(* PLC project MotionTest1, Higen MCL 1 *)
(* stored: creationDateTime 2012-01-06T15:20:13, modificationDateTime 2013-07-14T17:27:56 *)

FUNCTION_BLOCK wxgetval
  VAR
    getpy : python_gear;
    latch : SR;
  END_VAR
  VAR_INPUT
    name : STRING;
  END_VAR
  VAR_OUTPUT
    val : BOOL;
  END_VAR
  VAR  (* added by the conversion: wires and edge detectors of the diagram *)
    _EQ41_ENO : BOOL;
    _EQ41_OUT : BOOL;
    _EQ3_ENO : BOOL;
    _EQ3_OUT : BOOL;
  END_VAR

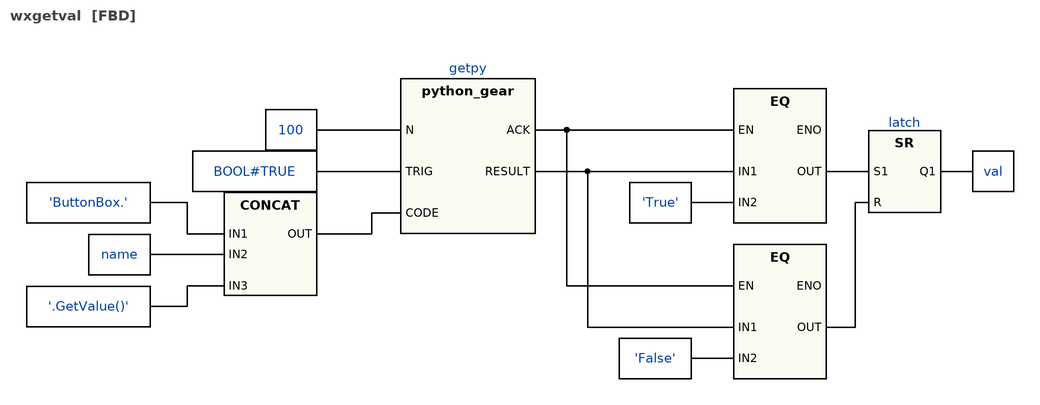
(* FBD diagram, written out as Structured Text *)
getpy(N := 100, TRIG := BOOL#TRUE, CODE := CONCAT('ButtonBox.', name, '.GetValue()'));
_EQ41_OUT := EQ(EN := getpy.ACK, IN1 := getpy.RESULT, IN2 := 'True', ENO => _EQ41_ENO);
_EQ3_OUT := EQ(EN := getpy.ACK, IN1 := getpy.RESULT, IN2 := 'False', ENO => _EQ3_ENO);
latch(S1 := _EQ41_OUT, R := _EQ3_OUT);
val := latch.Q1;
END_FUNCTION_BLOCK

(* -- *)
PROGRAM main
  VAR
    Done : BOOL;
    Axis : AXIS_REF;
    mPn : LREAL;
    mVn : LREAL;
    bt1 : wxgetval;
    Block1 : wxgetval;
    Block6 : wxgetval;
    MC_Sim0 : MC_Sim;
    MC_Power0 : MC_Power;
    MC_ReadActualPosition0 : MC_ReadActualPosition;
    MC_SetPosition0 : MC_SetPosition;
    MC_MoveAbsolute0 : MC_MoveAbsolute;
    Output : MC_OUTPUT_REF;
    OutputBits : DWORD;
    Track1 : BOOL;
    Track2 : BOOL;
    Track3 : BOOL;
    Velocity : LREAL := 1000.0;
    TrackList : MC_TRACK_REF;
    CamSwitchList : MC_CAMSWITCH_REF;
    MC_TRACK_REF_FROM_CSV0 : MC_TRACK_REF_FROM_CSV;
    MC_CAMSWITCH_REF_FROM_CSV0 : MC_CAMSWITCH_REF_FROM_CSV;
    MC_DigitalCamSwitch0 : MC_DigitalCamSwitch;
    MC_CreateOutput0 : MC_CreateOutput;
    MC_ReadActualVelocity0 : MC_ReadActualVelocity;
    MC_ReadOutputBits0 : MC_ReadOutputBits;
    MC_MoveAbsolute1 : MC_MoveAbsolute;
    MC_MoveAbsolute2 : MC_MoveAbsolute;
    MC_MoveAbsolute3 : MC_MoveAbsolute;
    MC_MoveAbsolute4 : MC_MoveAbsolute;
    MC_MoveAbsolute5 : MC_MoveAbsolute;
    MC_ReadOutputBit0 : MC_ReadOutputBit;
    MC_ReadOutputBit1 : MC_ReadOutputBit;
    MC_WriteParameter0 : MC_WriteParameter;
    MC_MoveAbsolute6 : MC_MoveAbsolute;
    MC_MoveAbsolute7 : MC_MoveAbsolute;
    MC_MoveAbsolute8 : MC_MoveAbsolute;
    MC_ReadOutputBit2 : MC_ReadOutputBit;
  END_VAR

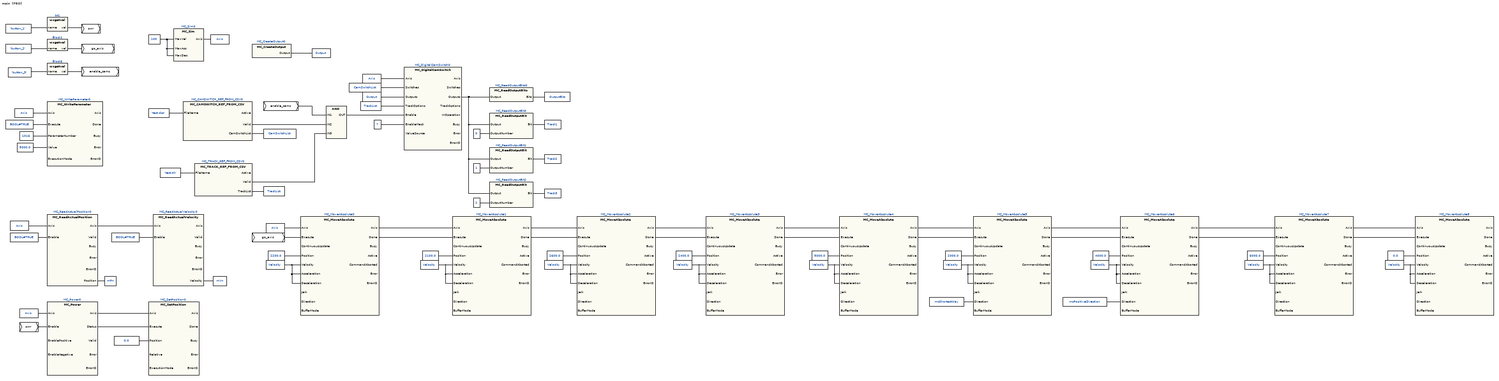
(* FBD diagram, written out as Structured Text *)
MC_Sim0(MaxVel := 100, MaxAcc := 100, MaxDec := 100);
Axis := MC_Sim0.Axis;
MC_CreateOutput0();
Output := MC_CreateOutput0.Output;
Block6(name := 'button_3');
MC_CAMSWITCH_REF_FROM_CSV0(FileName := 'test.dcs');
MC_TRACK_REF_FROM_CSV0(FileName := 'test.trk');
MC_DigitalCamSwitch0(Axis := Axis, Switches := CamSwitchList, Outputs := Output, TrackOptions := TrackList, Enable := Block6.val AND MC_CAMSWITCH_REF_FROM_CSV0.Valid AND MC_TRACK_REF_FROM_CSV0.Valid, EnableMask := 7);
MC_ReadOutputBits0(Output := MC_DigitalCamSwitch0.Outputs);
OutputBits := MC_ReadOutputBits0.Bits;
MC_ReadOutputBit0(Output := MC_DigitalCamSwitch0.Outputs, OutputNumber := 0);
Track1 := MC_ReadOutputBit0.Bit;
CamSwitchList := MC_CAMSWITCH_REF_FROM_CSV0.CamSwitchList;
MC_ReadOutputBit1(Output := MC_DigitalCamSwitch0.Outputs, OutputNumber := 1);
Track2 := MC_ReadOutputBit1.Bit;
TrackList := MC_TRACK_REF_FROM_CSV0.TrackList;
MC_ReadOutputBit2(Output := MC_DigitalCamSwitch0.Outputs, OutputNumber := 2);
Track3 := MC_ReadOutputBit2.Bit;
MC_ReadActualPosition0(Axis := Axis, Enable := BOOL#TRUE);
mPn := MC_ReadActualPosition0.Position;
MC_ReadActualVelocity0(Axis := MC_ReadActualPosition0.Axis, Enable := BOOL#TRUE);
mVn := MC_ReadActualVelocity0.Velocity;
bt1(name := 'button_1');
Block1(name := 'button_2');
MC_WriteParameter0(Axis := Axis, Execute := BOOL#TRUE, ParameterNumber := 1016, Value := 5000.0);
MC_MoveAbsolute0(Axis := Axis, Execute := Block1.val, Position := 2200.0, Velocity := Velocity, Acceleration := Velocity, Deceleration := Velocity);
MC_MoveAbsolute1(Axis := MC_MoveAbsolute0.Axis, Execute := MC_MoveAbsolute0.Done, Position := 2100.0, Velocity := Velocity, Acceleration := Velocity, Deceleration := Velocity);
MC_MoveAbsolute2(Axis := MC_MoveAbsolute1.Axis, Execute := MC_MoveAbsolute1.Done, Position := 2600.0, Velocity := Velocity, Acceleration := Velocity, Deceleration := Velocity);
MC_MoveAbsolute3(Axis := MC_MoveAbsolute2.Axis, Execute := MC_MoveAbsolute2.Done, Position := 2400.0, Velocity := Velocity, Acceleration := Velocity, Deceleration := Velocity);
MC_MoveAbsolute4(Axis := MC_MoveAbsolute3.Axis, Execute := MC_MoveAbsolute3.Done, Position := 5000.0, Velocity := Velocity, Acceleration := Velocity, Deceleration := Velocity);
MC_MoveAbsolute5(Axis := MC_MoveAbsolute4.Axis, Execute := MC_MoveAbsolute4.Done, Position := 2000.0, Velocity := Velocity, Acceleration := Velocity, Deceleration := Velocity, Direction := mcShortestWay);
MC_MoveAbsolute6(Axis := MC_MoveAbsolute5.Axis, Execute := MC_MoveAbsolute5.Done, Position := 4000.0, Velocity := Velocity, Acceleration := Velocity, Deceleration := Velocity, Direction := mcPositiveDirection);
MC_MoveAbsolute7(Axis := MC_MoveAbsolute6.Axis, Execute := MC_MoveAbsolute6.Done, Position := 6000.0, Velocity := Velocity, Acceleration := Velocity, Deceleration := Velocity);
MC_MoveAbsolute8(Axis := MC_MoveAbsolute7.Axis, Execute := MC_MoveAbsolute7.Done, Position := 0.0, Velocity := Velocity, Acceleration := Velocity, Deceleration := Velocity);
MC_Power0(Axis := Axis, Enable := bt1.val);
MC_SetPosition0(Axis := MC_Power0.Axis, Execute := MC_Power0.Status, Position := 0.0);
END_PROGRAM

CONFIGURATION conf
  RESOURCE res ON PLC
    TASK milisecond(INTERVAL := T#10ms, PRIORITY := 0);
    PROGRAM maininstance WITH milisecond : main;
  END_RESOURCE
END_CONFIGURATION
